TYPE ST_TestFunctionBlock :
STRUCT
	//pAddress : I_TestFunctionBlock;
	nNumberOfTests : UINT;
	aTestNames : ARRAY[0..100] OF T_MaxString;
	eTestFunctionBlockRunState : E_TestFunctionBlockRunState := E_TestFunctionBlockRunState.IDLE;
END_STRUCT
END_TYPE

(* stored: Version 1.1.0.1, ProductVersion 3.1.4022.12
   DUT ST_TestFunctionBlock: Id {13d3f096-dc15-407c-bd1a-874a6ea7d8e4} *)
